// Mitsubishi GX Works2 project: 시퀀스 자동동작, 수동동작   PLC: Q03UDV

PROGRAM MAIN
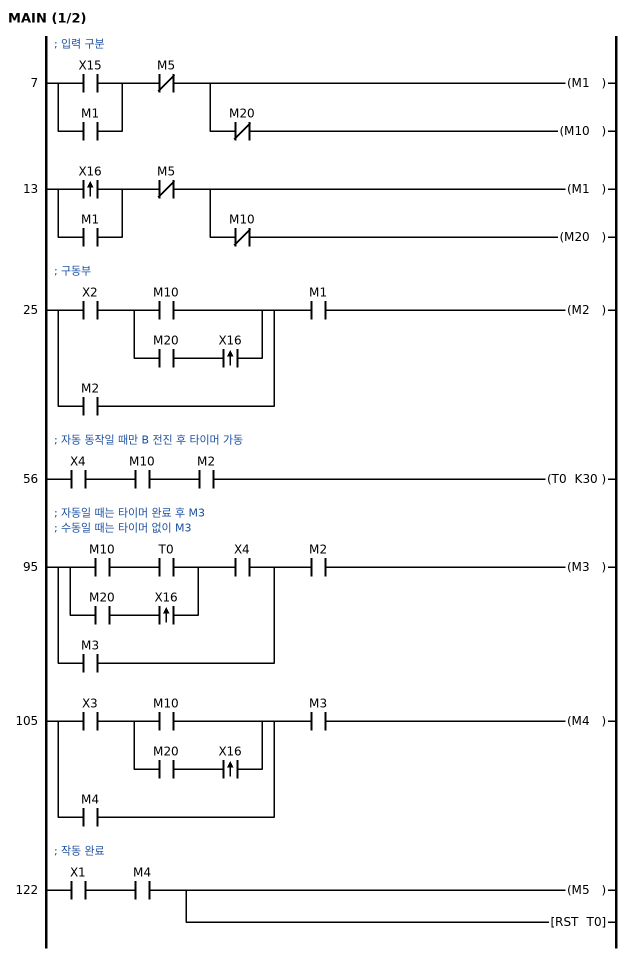
; 입력 구분
7     LD      X15
      OR      M1
      ANI     M5
      OUT     M1
      ANI     M20
      OUT     M10
13    LDP     X16
      OR      M1
      ANI     M5
      OUT     M1
      ANI     M10
      OUT     M20
; 구동부
25    LD      X2
      LD      M10
      LD      M20
      ANDP    X16
      ORB
      ANB
      OR      M2
      AND     M1
      OUT     M2
; 자동 동작일 때만 B 전진 후 타이머 가동
56    LD      X4
      AND     M10
      AND     M2
      OUT     T0 K30
; 자동일 때는 타이머 완료 후 M3
; 수동일 때는 타이머 없이 M3
95    LD      M10
      AND     T0
      LD      M20
      ANDP    X16
      ORB
      AND     X4
      OR      M3
      AND     M2
      OUT     M3
105   LD      X3
      LD      M10
      LD      M20
      ANDP    X16
      ORB
      ANB
      OR      M4
      AND     M3
      OUT     M4
; 작동 완료
122   LD      X1
      AND     M4
      OUT     M5
      RST     T0
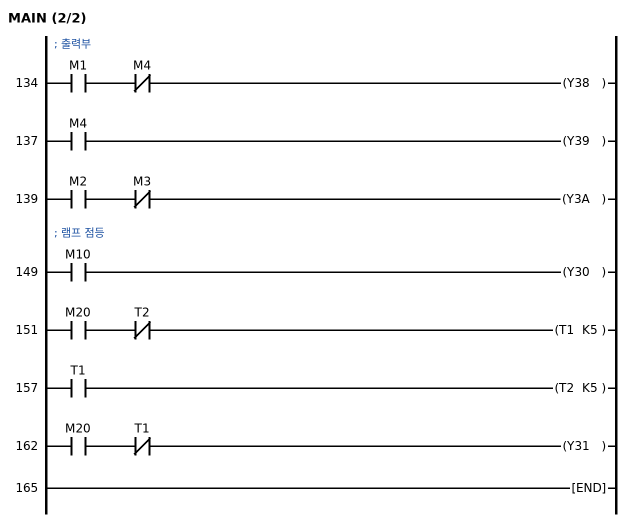
; 출력부
134   LD      M1
      ANI     M4
      OUT     Y38
137   LD      M4
      OUT     Y39
139   LD      M2
      ANI     M3
      OUT     Y3A
; 램프 점등
149   LD      M10
      OUT     Y30
151   LD      M20
      ANI     T2
      OUT     T1 K5
157   LD      T1
      OUT     T2 K5
162   LD      M20
      ANI     T1
      OUT     Y31
165   END
END_PROGRAM
